// TIA Portal V19 export
TYPE "type_materialParError"
// stored: Access Published
   STRUCT
      error : Bool;
   END_STRUCT;
END_TYPE
